FUNCTION_BLOCK FB_EndoscopeController
VAR_INPUT
END_VAR
VAR_OUTPUT
END_VAR
VAR
	// steering wheel parameter
	m_wheelRadius:LREAL;
	m_wheelHeight:ARRAY[1..2] OF LREAL;
	m_wheelCenter:ARRAY[1..2] OF Vec3d;
	
	// VF position control parameters
	m_VFPts :ARRAY[1..2] OF Vec3d;
	m_VFDeviation :ARRAY[1..2] OF Vec3d;
	m_lastVFDeviation :ARRAY[1..2] OF Vec3d;
	m_VFVel :ARRAY[1..2] OF Vec3d;
	m_VFVelLpf:ARRAY[1..2,1..3] OF FB_LowPassFilter;
	m_VFKp :LREAL := 500;
	m_VFKd :LREAL := 15;
	m_VFForce :ARRAY[1..2] OF Vec3d;
	
	// oritention control parameter
	m_rotTrackKp : LREAL := 200;
	m_maxTrackVel :LREAL := PI;
	m_jnt4AdjustKp : LREAL :=10;
	m_jnt4MaxVel :LREAL :=pi/3 ;
	m_linearVelLb :LREAL := 0.01;
	m_linearVelUb :LREAL :=0.1;	
	m_cartTrackVel :Vec3d;
	
	// master pose in monitor
	tmpVFPt :ARRAY[1..2] OF Vec3d;
	m_masterPoseInView :ARRAY[1..2] OF ST_Frame;
	
	// orientation deviation between master and slave when first enter control
	m_MSOriDeviation :ARRAY[1..2] OF Mat3d;
	m_firstIn : ARRAY[1..2] OF BOOL :=[TRUE, TRUE];
	
	// flag if the controller has finished all its jobs
	m_isFinished:BOOL:=FALSE;
	
	// controller execute time period
	m_timePeriod :LREAL:=0;
	
	// arm control data
	m_cmdJntPos :ARRAY[1..2] OF VEC7d;
	m_cmdJntVel :ARRAY[1..2] OF VEC7d;
	m_cmdJntAcc :ARRAY[1..2] OF VEC7d;
	m_cmdJntTrq :ARRAY[1..2] OF VEC7d;
	m_jntOPMode :ARRAY[1..2] OF Vec7i;
	m_jntEnableFlag :ARRAY[1..2] OF Vec7i;
	m_cmdCartPose :ARRAY[1..2] OF ST_Frame;
	m_cmdCartTwist :ARRAY[1..2] OF Vec6d;
	
	// joint4 dynamic limit 
	m_jntPosUb, m_jntPosLb:LREAL;
	
	// flag to follow instrument rotation
	m_slaveMatchFlag :ARRAY[1..2] OF BOOL;
	
END_VAR

// compute the desired joint position of joint 4-7 for orientation tracking
METHOD PROTECTED calcCmdJntPos : BOOL

VAR_IN_OUT CONSTANT
	i_teleSlaveArmIdx:ARRAY[1..2] OF E_MatchedSlaveArmIdx;
	i_shoulderPose:ARRAY[1..2] OF ST_Frame;
	i_masterArm :ARRAY[1..2] OF FB_MasterArm;
	i_slaveStatus : ST_SlaveStatus;
END_VAR
VAR 
	armIdx:INT;
	i,j : INT;
	
	cmdRotInMonitor,cmdRotInArm :Mat3d;
	invRot:Mat3d;
	
	rotT,rotErr:Mat3d;
	angle : LREAL;
	axis,localAxis :Vec3d;
	oriJaco:Mat3d;
	oriJacoInv:Mat3d;
	cartTrackVel:Vec3d;
	jntTrackVel:Vec3d;
	
END_VAR
FOR armIdx:=1 TO 2 DO
	// arm position is compliant
	m_cmdCartPose[armIdx].m_pos:= i_masterArm[armIdx].curCartPose.m_pos;
	FOR i:=1 TO 3 DO 
		m_cmdJntPos[armIdx][i]:=i_masterArm[armIdx].curJntPos[i];
		m_cmdJntVel[armIdx][i]:=i_masterArm[armIdx].curJntVel[i];
	END_FOR
	
	
	// update command oritentation if corresponding slave arm is in SlaveArmState_InstruReady state
	IF i_slaveStatus.m_armState[i_teleSlaveArmIdx[armIdx]] = SlaveArmState_Adjust OR
		NOT(i_slaveStatus.m_instruStauts[i_teleSlaveArmIdx[armIdx]].m_ready) THEN
		m_slaveMatchFlag[armIdx] :=FALSE;
	END_IF
	IF m_slaveMatchFlag[armIdx] THEN
		// command rotation in monitor
		cmdRotInMonitor := i_slaveStatus.m_curArmPose[i_teleSlaveArmIdx[armIdx]].m_rot;
		
		// command rotation in master arm base
		matTranspose(i_shoulderPose[armIdx].m_rot, invRot);
		matMultiply(invRot, cmdRotInMonitor, cmdRotInArm);
		
		// handle orientation deviation for the first time in
		IF m_firstIn[armIdx] THEN
			m_firstIn[armIdx] := FALSE;
			matTranspose(cmdRotInArm, invRot);
			matMultiply(invRot, i_masterArm[armIdx].curCartPose.m_rot,m_MSOriDeviation[armIdx]);
		END_IF
		
		matMultiply(cmdRotInArm, m_MSOriDeviation[armIdx],m_cmdCartPose[armIdx].m_rot);
	END_IF

	// compute cartesian tracking velocity
	matTranspose(i_masterArm[armIdx].simCartPose.m_rot, rotT);
	matMultiply(rotT, m_cmdCartPose[armIdx].m_rot, rotErr);
	rot2AngAxis(rotErr, angle=>angle,axis=>localAxis);
	matMultiVec(i_masterArm[armIdx].simCartPose.m_rot, localAxis, axis);
	vecMultiNum(axis, LIMIT(-m_maxTrackVel, angle*m_rotTrackKp, m_maxTrackVel), cartTrackVel);
	m_cartTrackVel :=cartTrackVel;
	
	// compute pinv of orientation jacobian
	FOR i:=1 TO 3 DO
		FOR j:=1 TO 3 DO
			oriJaco[i,j]:=i_masterArm[armIdx].simJaco[i+3,j+4];
		END_FOR
	END_FOR
	invMat3(oriJaco, oriJacoInv);
	matMultiVec(oriJacoInv, cartTrackVel, jntTrackVel);
	
	// update final command joint position and velocity
	FOR i :=5 TO 7 DO 
		m_cmdJntVel[armIdx][i]:=jntTrackVel[i-4];
		m_cmdJntPos[armIdx][i]:=m_cmdJntPos[armIdx][i]+m_cmdJntVel[armIdx][i]*g_armCtrlCycleTime;
	END_FOR
	
//	// compute pinv of orientation jacobian
//	FOR i:=1 TO 3 DO
//		FOR j:=1 TO 4 DO
//			oriJaco[i,j]:=i_masterArm[armIdx].simJaco[i+3,j+3];
//		END_FOR
//	END_FOR
//	matTranspose(oriJaco, oriJt);
//	matMultiply(oriJaco ,oriJt , oriJJt);
//	invMat3(oriJJt, oriJJtInv);
//	matMultiply(oriJt, oriJJtInv, oriJPinv);
//	matMultiVec(oriJpinv, cartTrackVel, jntTrackVel);
	
//	// calculate nullspace
//	matMultiply(oriJPinv, oriJaco, JpinvJ);
//	matSub(eye4d , JpinvJ, nullJ);
	
//	// redundant velocity
//	jnt4TrackVel:=calcRedunVel(i_masterArm[armIdx]);
//	redunCtrlVel[1]:=nullJ[1,1]*jnt4TrackVel;
//	redunCtrlVel[2]:=nullJ[2,1]*jnt4TrackVel;
//	redunCtrlVel[3]:=nullJ[3,1]*jnt4TrackVel;
//	redunCtrlVel[4]:=nullJ[4,1]*jnt4TrackVel;
	
//	// update final command joint position and velocity
//	FOR i :=1 TO 4 DO 
//		m_cmdJntVel[armIdx][i+3]:=jntTrackVel[i]+redunCtrlVel[i];
//		m_cmdJntPos[armIdx][i+3]:=m_cmdJntPos[armIdx][i+3]+m_cmdJntVel[armIdx][i+3]*g_armCtrlCycleTime;
//	END_FOR
	
	// redundant control
	calcRedunMotion(i_masterArm[armIdx]);

END_FOR
END_METHOD

// compute the desired joint torque of joint 1-3 for intuitive force guiding
METHOD PROTECTED calcCmdJntTrq : BOOL

VAR_IN_OUT CONSTANT
	i_teleSlaveArmIdx:ARRAY[1..2] OF E_MatchedSlaveArmIdx;
	i_shoulderPose:ARRAY[1..2] OF ST_Frame;
	i_masterArm :ARRAY[1..2] OF FB_MasterArm;
	i_slaveStatus : ST_SlaveStatus;
END_VAR

VAR 
	
	armIdx :INT;
	i,j :INT;
	kpForce, kdForce :Vec3d;
	jntTrq :Vec3d;
	posJaco, posJacoT :Mat3d;
	trqScale :LREAL;
END_VAR
m_cmdJntTrq[1] := g_zeroVec7d;
m_cmdJntTrq[2] := g_zeroVec7d;

// compute cuurent VF parameters
steeringWheelCalc(i_shoulderPose, i_masterArm);

// compute VF motion velocity
FOR armIdx:=1 TO 2 DO
	vecSub(m_lastVFDeviation[armIdx],m_VFDeviation[armIdx], m_VFVel[armIdx]);
	vecSelfMultiNum(m_VFVel[armIdx], g_armCtrlFreq);
	FOR j:=1 TO 3 DO 
		m_VFVel[armIdx][j] := m_VFVelLpf[armIdx,j].run(m_VFVel[armIdx][j]);
	END_FOR
	
	m_lastVFDeviation[armIdx] := m_VFDeviation[armIdx];
END_FOR

// compute VF force
FOR armIdx:=1 TO 2 DO
	vecMultiNum(m_VFDeviation[armIdx], m_VFKp, kpForce);
	vecMultiNum(m_VFVel[armIdx], m_VFKd, kdForce);
	vecSub(kpForce, kdForce, m_VFForce[armIdx]);
END_FOR

// compute joint space torque
FOR armIdx:=1 TO 2 DO 
	FOR i :=1 TO  3 DO
		FOR j:=1 TO 3 DO
			posJaco[i,j]:= i_masterArm[armIdx].jaco[i,j];
		END_FOR
	END_FOR
	matTranspose(posJaco, posJacoT);
	matMultiVec(posJacoT, m_VFForce[armIdx], jntTrq);
	
	// scale joint troque
	trqScale := 1;
	FOR i:=1 TO 3 DO 
		trqScale:=MAX(trqScale, ABS(jntTrq[i]/GVL_ArmJointParameters.g_jntMaxTrq[i]));
	END_FOR
	
	m_cmdJntTrq[armIdx][1]:=jntTrq[1]/trqScale;
	m_cmdJntTrq[armIdx][2]:=jntTrq[2]/trqScale;
	m_cmdJntTrq[armIdx][3]:=jntTrq[3]/trqScale;
END_FOR
END_METHOD

METHOD PROTECTED calcRedunMotion : LREAL
VAR_IN_OUT CONSTANT
	i_masterArm :FB_MasterArm;
END_VAR

VAR 
	j6Bias,j5Bias :LREAL;
	velScale :LREAL;
	linearVel :Vec3d;
	curJntPos : Vec7d;
	jnt4LinkPos :LREAL;
	armJaco :Mat3d;
	armJntVel, armW:Vec3d;
	wristJaco, wristJacoInv:Mat3d;
	wristJntVel:Vec3d;
	i,j :INT;
	cmdFFJntVel:LREAL;
	coupleJntVel:LREAL;
END_VAR
// compute desired joint4 link position
curJntPos :=  i_masterArm.cmdJntPos;
jnt4LinkPos:=i_masterArm.jnt4MotorToLink(curJntPos[2],curJntPos[3],curJntPos[4]);
IF 1= i_masterArm.armIdx THEN
	j6Bias :=curJntPos[6]+PI/2;
ELSE 
	j6Bias := curJntPos[6]-PI/2;
END_IF

// scale based on joint5 position
j5Bias :=  LIMIT (0, ABS(curJntPos[5] -pi), pi/2);
j6Bias := j6Bias * ABS(COS(j5Bias));

// scale based on linear velocity
linearVel[1]:=i_masterArm.curCartTwist[1];
linearVel[2]:=i_masterArm.curCartTwist[2];
linearVel[3]:=i_masterArm.curCartTwist[3];
velScale :=LIMIT(0, (norm(linearVel)-m_linearVelLb)/(m_linearVelUb-m_linearVelLb),1.0);

m_cmdJntVel[i_masterArm.armIdx][4] := LIMIT(-m_jnt4MaxVel, -j6Bias * m_jnt4AdjustKp * velScale ,m_jnt4MaxVel);

// compute feedforward velocity to compensate joint1 motion
FOR i :=1 TO 3 DO
	FOR j:=1 TO 3 DO 
		armJaco[i,j]:= i_masterArm.jaco[i+3,j];
		wristJaco[i,j]:= i_masterArm.jaco[i+3,j+4];
	END_FOR
END_FOR
InvMat3(wristJaco, wristJacoInv);
armJntVel:=g_zeroVec3d;
armJntVel[1]:=i_masterArm.curJntVel[1];
matMultiVec(armJaco, armJntVel, armW);
matMultiVec(wristJacoInv, armW, wristJntVel);
cmdFFJntVel:=wristJntVel[2];
m_cmdJntVel[i_masterArm.armIdx][4]:=m_cmdJntVel[i_masterArm.armIdx][4]+cmdFFJntVel;

// joint limit
IF (m_cmdJntVel[i_masterArm.armIdx][4] > 0 AND jnt4LinkPos+m_cmdJntVel[i_masterArm.armIdx][4] * g_armCtrlCycleTime > GVL_ArmJointParameters.g_maxJntPos[i_masterArm.armIdx,4]-GVL_ArmJointParameters.g_jntLimitBuffer)
	 OR ( m_cmdJntVel[i_masterArm.armIdx][4] <0 AND  jnt4LinkPos +m_cmdJntVel[i_masterArm.armIdx][4] * g_armCtrlCycleTime< GVL_ArmJointParameters.g_minJntPos[i_masterArm.armIdx,4]+GVL_ArmJointParameters.g_jntLimitBuffer) THEN
	 m_cmdJntVel[i_masterArm.armIdx][4] :=0;
END_IF
m_cmdJntPos[i_masterArm.armIdx][4]:=m_cmdJntPos[i_masterArm.armIdx][4]+m_cmdJntVel[i_masterArm.armIdx][4]*g_armCtrlCycleTime;

// compute feedforward velocity to compensate joint1 motion
coupleJntVel := i_masterArm.curJntVel[2]-i_masterArm.curJntVel[3];
m_cmdJntVel[i_masterArm.armIdx][4]:= m_cmdJntVel[i_masterArm.armIdx][4] + coupleJntVel;
m_cmdJntPos[i_masterArm.armIdx][4]:=m_cmdJntPos[i_masterArm.armIdx][4]+coupleJntVel*g_armCtrlCycleTime;
// position limit check
m_jntPosUb:=i_masterArm.jnt4LinkToMotor(i_masterArm.curJntPos[2],i_masterArm.curJntPos[3],
						 GVL_ArmJointParameters.g_maxJntPos[i_masterArm.armIdx,4]-GVL_ArmJointParameters.g_jntLimitBuffer);
m_jntPosLb:=i_masterArm.jnt4LinkToMotor(i_masterArm.curJntPos[2],i_masterArm.curJntPos[3],
						 GVL_ArmJointParameters.g_minJntPos[i_masterArm.armIdx,4]+GVL_ArmJointParameters.g_jntLimitBuffer);
IF m_cmdJntPos[i_masterArm.armIdx][4] >=m_jntPosUb OR m_cmdJntPos[i_masterArm.armIdx][4]<m_jntPosLb THEN
	m_cmdJntVel[i_masterArm.armIdx][4]:=0;
	m_cmdJntPos[i_masterArm.armIdx][4]:=LIMIT(m_jntPosLb,m_cmdJntPos[i_masterArm.armIdx][4],m_jntPosUb);
END_IF
END_METHOD

// override this function in each exact controller
// NOTICE: set joint control mode here, and do some initialization if needed
METHOD PUBLIC init : BOOL
VAR_IN_OUT CONSTANT
	i_shoulderPose:ARRAY[1..2] OF ST_Frame;
	i_masterArm :ARRAY[1..2] OF FB_MasterArm;
END_VAR
VAR_IN_OUT 
	r_masterArmCtrlCmd :ARRAY[1..2] OF ST_ArmCtrlCmds;
END_VAR
VAR
	i,j:INT;
END_VAR
m_timePeriod:=0;
FOR i:=1 TO 2 DO 
	m_jntEnableFlag[i] :=g_onesVec7i;
	m_jntOPMode[i][1] := DriverOPMode_Trq;
	m_jntOPMode[i][2] := DriverOPMode_Trq;
	m_jntOPMode[i][3] := DriverOPMode_Trq;
	m_jntOPMode[i][4] := DriverOPMode_PosTrq;
	m_jntOPMode[i][5] := DriverOPMode_PosTrq;
	m_jntOPMode[i][6] := DriverOPMode_PosTrq;
	m_jntOPMode[i][7] := DriverOPMode_PosTrq;
	m_cmdCartPose[i]:=i_masterArm[i].curCartPose;
	m_cmdCartTwist[i]:=g_zeroVec6d;
	m_cmdJntPos[i]:=i_masterArm[i].curJntPos;
	m_cmdJntVel[i]:=g_zeroVec7d;
	m_cmdJntAcc[i]:=g_zeroVec7d;
	m_cmdJntTrq[i]:=g_zeroVec7d;
	
	r_masterArmCtrlCmd[i].m_jntEnableFlag :=m_jntEnableFlag[i];
	r_masterArmCtrlCmd[i].m_cmdCartPose:=m_cmdCartPose[i];
	r_masterArmCtrlCmd[i].m_cmdCartTwist:=m_cmdCartTwist[i];
	r_masterArmCtrlCmd[i].m_cmdJntPos:=m_cmdJntPos[i];
	r_masterArmCtrlCmd[i].m_cmdJntVel:=m_cmdJntVel[i];
	r_masterArmCtrlCmd[i].m_cmdJntAcc:=m_cmdJntAcc[i];
	r_masterArmCtrlCmd[i].m_cmdJntTrq:=m_cmdJntTrq[i];
	r_masterArmCtrlCmd[i].m_jntOPMode:=m_jntOPMode[i];
	
	m_lastVFDeviation[i] := g_zeroVec3d;
	
	m_firstIn[i] := TRUE;
	m_MSOriDeviation[i] := g_eye3d;
	
	// filter init
	FOR j:=1 TO 3 DO 
		m_VFVelLpf[i,j].init(1, g_curJntVelLpfCutoffFreq, g_armCtrlFreq);
	END_FOR
	
	m_slaveMatchFlag[i] :=true;

END_FOR

steeringWheelInit(i_shoulderPose, i_masterArm);
END_METHOD

// TODO: corner case that two arm tips coincide on z axis need to be handle
METHOD run : BOOL

VAR_IN_OUT CONSTANT
	i_teleSlaveArmIdx:ARRAY[1..2] OF E_MatchedSlaveArmIdx;
	i_shoulderPose:ARRAY[1..2] OF ST_Frame;
	i_masterArm :ARRAY[1..2] OF FB_MasterArm;
	i_slaveStatus : ST_SlaveStatus;
END_VAR
VAR_IN_OUT 
	r_masterArmCtrlCmd :ARRAY[1..2] OF ST_ArmCtrlCmds;
END_VAR
VAR
	i:INT;
END_VAR
IF m_isFinished THEN
	RETURN;
END_IF

// check if arm enabled
IF NOT(i_masterArm[1].isEnabled(m_jntEnableFlag[1])) OR NOT(i_masterArm[2].isEnabled(m_jntEnableFlag[2]))  THEN
	RETURN;
END_IF

// calculate command joint position--Motion control
calcCmdJntPos(i_teleSlaveArmIdx, i_shoulderPose, i_masterArm,i_slaveStatus);

// calculate command joint torque -- Force control
calcCmdJntTrq(i_teleSlaveArmIdx, i_shoulderPose, i_masterArm,i_slaveStatus);

// update commands to arm
FOR i:=1 TO 2 DO 
	r_masterArmCtrlCmd[i].m_cmdJntPos:=m_cmdJntPos[i];
	r_masterArmCtrlCmd[i].m_cmdJntTrq:=m_cmdJntTrq[i];
END_FOR

// update time period
m_timePeriod := m_timePeriod+g_armCtrlCycleTime;
END_METHOD

METHOD PROTECTED steeringWheelCalc : BOOL
VAR_IN_OUT CONSTANT
	i_shoulderPose:ARRAY[1..2] OF ST_Frame;
	i_masterArm :ARRAY[1..2] OF FB_MasterArm;
END_VAR
VAR
	tipCenter :Vec3d;
	i:INT;

	rotT :Mat3d;
	VFDeviationInView:Vec3d;
END_VAR
// master pose in view coordinate
m_masterPoseInView[1] := transform(i_shoulderPose[1],  i_masterArm[1].curCartPose);
m_masterPoseInView[2] := transform(i_shoulderPose[2],  i_masterArm[2].curCartPose);

// master tip center 
vecAdd(m_masterPoseInView[1].m_pos, m_masterPoseInView[2].m_pos, tipCenter);
vecSelfMultiNum(tipCenter,0.5);

FOR i:=1 TO 2 DO 
	// steering wheel center 
	m_wheelCenter[i]:=tipCenter;
	m_wheelCenter[i][3]:=m_wheelCenter[i][3]+m_wheelHeight[i];
	
	// compute current virtual fixture points on wheel 
	vecSub(m_masterPoseInView[i].m_pos, m_wheelCenter[i], tmpVFPt[i]);
	tmpVFPt[i][3]:=0;
	IF NOT(normalize(tmpVFPt[i])) THEN
		steeringWheelCalc := FALSE;
		RETURN;
	END_IF
	vecSelfMultiNum(tmpVFPt[i], m_wheelRadius);
	vecAdd(m_wheelCenter[i], tmpVFPt[i], m_VFPts[i]);
	
	// compute current deviation from VF points in shoulder coordinate
	vecSub(m_VFPts[i], m_masterPoseInView[i].m_pos, VFDeviationInView);
	matTranspose(i_shoulderPose[i].m_rot , rotT);
	matMultiVec(rotT, VFDeviationInView, m_VFDeviation[i]);

END_FOR
END_METHOD

METHOD PROTECTED steeringWheelInit : BOOL
VAR_IN_OUT CONSTANT
	i_shoulderPose:ARRAY[1..2] OF ST_Frame;
	i_masterArm :ARRAY[1..2] OF FB_MasterArm;
END_VAR
VAR
	tipDis,tipCenter :Vec3d;
END_VAR
// master pose in view coordinate
m_masterPoseInView[1] := transform(i_shoulderPose[1],  i_masterArm[1].curCartPose);
m_masterPoseInView[2] := transform(i_shoulderPose[2],  i_masterArm[2].curCartPose);

// master tip height relative to center 
vecAdd(m_masterPoseInView[1].m_pos, m_masterPoseInView[2].m_pos, tipCenter);
vecSelfMultiNum(tipCenter,0.5);
m_wheelHeight[1] :=m_masterPoseInView[1].m_pos[3] -  tipCenter[3];
m_wheelHeight[2] :=m_masterPoseInView[2].m_pos[3] -  tipCenter[3];

// master tip distance  relative to center 
vecSub(m_masterPoseInView[1].m_pos, m_masterPoseInView[2].m_pos, tipDis);
tipDis[3] := 0;
m_wheelRadius :=norm(tipDis)/2.0;
END_METHOD

END_FUNCTION_BLOCK

(* stored: Version 1.1.0.1, ProductVersion 3.1.4024.12
   POU FB_EndoscopeController: Id {311b6261-a50e-45fe-88ed-e8188e25e8c2}, SpecialFunc None
   Method calcCmdJntPos: Id {010ad3dd-bcc4-454c-abf2-f1c15ea59de0}
   Method calcCmdJntTrq: Id {b8016091-c8e3-4690-ae2f-cd184a2d59dd}
   Method calcRedunMotion: Id {e5f2707d-71a6-4ce7-a32b-89a14f84d3b2}
   Method init: Id {4f8bfc3d-09c7-4a85-920c-1b402f5c5a84}
   Method run: Id {b5febb70-d533-42f5-b7c9-4e139b9a0211}
   Method steeringWheelCalc: Id {32a6a63f-edcb-492d-b3a3-3fd59305455a}
   Method steeringWheelInit: Id {e55932b2-6de1-40a4-bfce-4f83b95e9fbb} *)
